PROGRAM PRG_10_TempHumidAnalytics
VAR
	TempSensor								: GenericSensor;
	HumiditySensor							: GenericSensor;
	
	TempSensorPostHTTP						: HttpPost;
	HumiditySensorPostHTTP					: HttpPost;
END_VAR

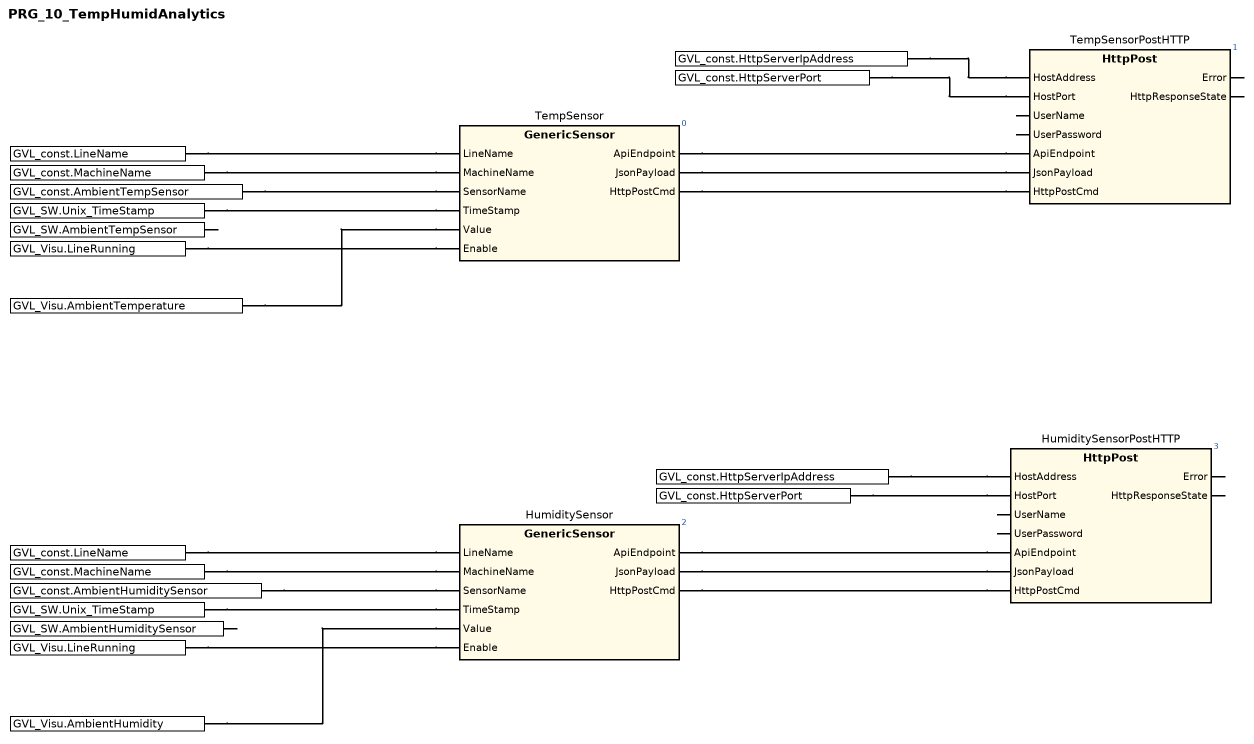
TempSensor(
    LineName := GVL_const.LineName,
    MachineName := GVL_const.MachineName,
    SensorName := GVL_const.AmbientTempSensor,
    TimeStamp := GVL_SW.Unix_TimeStamp,
    Value := GVL_Visu.AmbientTemperature,
    Enable := GVL_Visu.LineRunning); // GenericSensor
TempSensorPostHTTP(
    HostAddress := GVL_const.HttpServerIpAddress,
    HostPort := GVL_const.HttpServerPort,
    ApiEndpoint := TempSensor.ApiEndpoint,
    JsonPayload := TempSensor.JsonPayload,
    HttpPostCmd := TempSensor.HttpPostCmd); // HttpPost
HumiditySensor(
    LineName := GVL_const.LineName,
    MachineName := GVL_const.MachineName,
    SensorName := GVL_const.AmbientHumiditySensor,
    TimeStamp := GVL_SW.Unix_TimeStamp,
    Value := GVL_Visu.AmbientHumidity,
    Enable := GVL_Visu.LineRunning); // GenericSensor
HumiditySensorPostHTTP(
    HostAddress := GVL_const.HttpServerIpAddress,
    HostPort := GVL_const.HttpServerPort,
    ApiEndpoint := HumiditySensor.ApiEndpoint,
    JsonPayload := HumiditySensor.JsonPayload,
    HttpPostCmd := HumiditySensor.HttpPostCmd); // HttpPost
// GVL_SW.AmbientTempSensor: input not connected
// GVL_SW.AmbientHumiditySensor: input not connected

END_PROGRAM

(* stored: Version 1.1.0.1, ProductVersion 3.1.4024.15
   POU PRG_10_TempHumidAnalytics: Id {71aa9778-4091-4bf1-b573-d9e4e399eb71}, SpecialFunc None *)
